FUNCTION_BLOCK Pusher_Element (* Basic Function Block Type *)
  (* Standard: 61499-2 *)
  (* Version 0.0, 21/06/2022, Lernfabrik, WBK hackaton, Template *)
  PACKAGE Main;
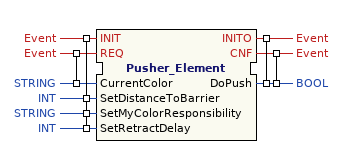
  EVENT_INPUT
    INIT WITH SetDistanceToBarrier, SetMyColorResponsibility, SetRetractDelay; (* Initialization Request *)
    REQ WITH CurrentColor; (* Normal Execution Request *)
  END_EVENT
  EVENT_OUTPUT
    INITO WITH DoPush; (* Initialization Confirm *)
    CNF WITH DoPush; (* Execution Confirmation *)
  END_EVENT
  VAR_INPUT
    CurrentColor : STRING; (* Color of the Element Currently at the last Barrier *)
    SetDistanceToBarrier : INT;
    SetMyColorResponsibility : STRING := 'Green'; (* Setup the Color I am responsible for *)
    SetRetractDelay : INT;
  END_VAR
  VAR_OUTPUT
    DoPush : BOOL; (* Output event qualifier *)
  END_VAR
  VAR
    DistanceToBarrier : INT; (* Distance in Ticks to the Exit Barrier (Nr. 2) *)
    RetractDelay : INT; (* Time until the Pusher retrackts after pushing our thing away *)
    MyColorResponsibility : STRING := 'Green'; (* Elements of which color should I push out? *)
    InOutState : BOOL := FALSE; (* 0 = Back 1 = Pusher out *)
    RemainingTicks : INT;
    Activated : BOOL := FALSE;
  END_VAR
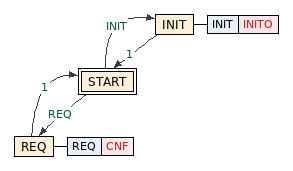
  EC_STATES
    START; (* Initial State *)
    INIT : INIT -> INITO; (* Initialization *)
    REQ : REQ -> CNF; (* Normal execution *)
  END_STATES
  EC_TRANSITIONS
    START TO INIT := INIT;
    INIT TO START := 1;
    START TO REQ := REQ;
    REQ TO START := 1;
  END_TRANSITIONS
  ALGORITHM INIT IN ST: (* Initialization algorithm *)
InOutState := 0;
RetractDelay := 1;
MyColorResponsibility := SetMyColorResponsibility;
DistanceToBarrier := SetDistanceToBarrier;
(* ToDo: Retract Once *)
  END_ALGORITHM
  ALGORITHM REQ IN ST: (* Normally executed algorithm *)
IF MyColorResponsibility = CurrentColor THEN
	RemainingTicks := DistanceToBarrier;
	Activated := 1;
	(* What happens if the same color comes twice in a cycle? -> Oh, oh*)
END_IF;

RemainingTicks := RemainingTicks - 1;
IF RemainingTicks < 1 AND RemainingTicks > -10 THEN
		DoPush := 1;
		Activated := 0;
		RemainingTicks := -10;

END_IF;
  END_ALGORITHM
END_FUNCTION_BLOCK
